// Mitsubishi GX Works2 project: q8   PLC: Q02/Q02H

PROGRAM MAIN
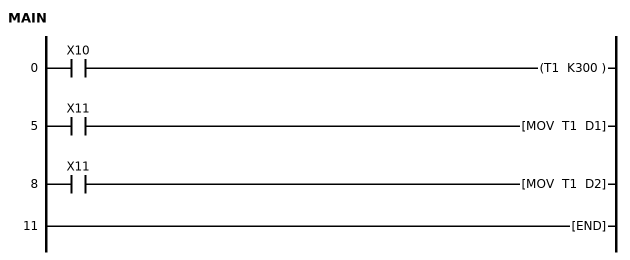
0     LD      X10
      OUT     T1 K300
5     LD      X11
      MOV     T1 D1
8     LD      X11
      MOV     T1 D2
11    END
END_PROGRAM
